// TIA Portal project "Project11" (V17)

(* hardware
DEVICE "S7-1200 station_1"  S7-1200 Station
   slot 0: "Rack_0"  S7-1200 Rack  Rack  V1.0
   slot 1: "PLC_1"  CPU 1214C AC/DC/Rly  6ES7 214-1BG40-0XB0  V4.2
*)

// ===== PLC "PLC_1"  CPU 1214C AC/DC/Rly =====

VAR_GLOBAL   // PLC tag table "Default tag table"
   "Tag_1" AT %M0.0 : Bool;
   "Tag_2" AT %M0.1 : Bool;
   "Tag_3" AT %M0.2 : Bool;
   "Tag_4" AT %M1.0 : Bool;
   "Tag_5" AT %M1.1 : Bool;
   "Tag_6" AT %M1.2 : Bool;
END_VAR

DATA_BLOCK "test1_DB"   // DB1
{ S7_Optimized_Access := 'TRUE' }
VERSION : 0.1
// stored: InstanceOfName test1
"test1"
BEGIN
END_DATA_BLOCK

FUNCTION_BLOCK "test1"   // FB1, LAD
{ S7_Optimized_Access := 'TRUE' }
VERSION : 0.1
   VAR_INPUT
      start : Bool;
      stop : Bool;
   END_VAR
   VAR_OUTPUT
      output : Bool;
   END_VAR
   VAR
      m1 : Bool;
   END_VAR
BEGIN

REGION Network 1
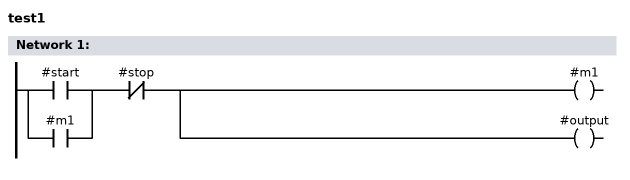
   RUNG wire#powerrail
      Contact( #start )
      wire#w1
      I_Contact( #stop )
      wire#w2
      Coil( #m1 )
   END_RUNG
   RUNG wire#powerrail
      Contact( #m1 )
   END_RUNG wire#w1
   RUNG wire#w2
      Coil( #output )
   END_RUNG
   // the same network as SCL:
   #m1 := (#start OR #m1) AND NOT #stop;
   #output := #m1;
END_REGION
END_FUNCTION_BLOCK

FUNCTION "test" : Void   // FC1, LAD
{ S7_Optimized_Access := 'TRUE' }
VERSION : 0.1
   VAR_INPUT
      start : Bool;
      stop : Bool;
   END_VAR
   VAR_OUTPUT
      output : Bool;
   END_VAR
   VAR_TEMP
      m1 : Bool;
   END_VAR
BEGIN

REGION Network 1
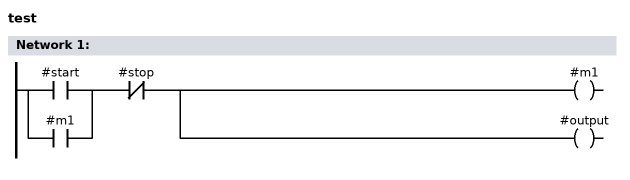
   RUNG wire#powerrail
      Contact( #start )
      wire#w1
      I_Contact( #stop )
      wire#w2
      Coil( #m1 )
   END_RUNG
   RUNG wire#powerrail
      Contact( #m1 )
   END_RUNG wire#w1
   RUNG wire#w2
      Coil( #output )
   END_RUNG
   // the same network as SCL:
   #m1 := (#start OR #m1) AND NOT #stop;
   #output := #m1;
END_REGION
END_FUNCTION

ORGANIZATION_BLOCK "Main"   // OB1, LAD, ProgramCycle
TITLE = "Main Program Sweep (Cycle)"
{ S7_Optimized_Access := 'TRUE' }
VERSION : 0.1
   VAR_INPUT
      Initial_Call : Bool;   // Initial call of this OB
      Remanence : Bool;   // =True, if remanent data are available
   END_VAR
BEGIN

REGION Network 1
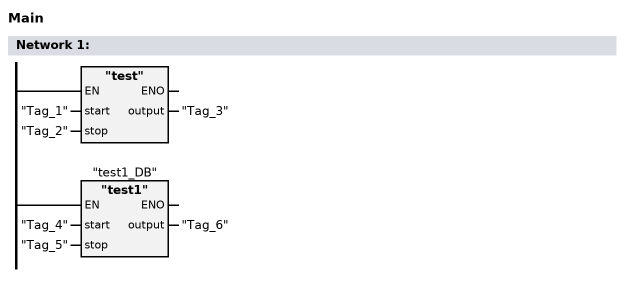
   RUNG wire#powerrail
      "test"(start := "Tag_1", stop := "Tag_2", output => "Tag_3")
   END_RUNG
   RUNG wire#powerrail
      "test1_DB"(start := "Tag_4", stop := "Tag_5", output => "Tag_6")
   END_RUNG
   // the same network as SCL:
   "test"(start := "Tag_1", stop := "Tag_2", output => "Tag_3");
   "test1_DB"(start := "Tag_4", stop := "Tag_5", output => "Tag_6");   // "test1"
END_REGION
END_ORGANIZATION_BLOCK